{attribute 'qualified_only'}
VAR_GLOBAL CONSTANT
	cuiNrChannel		: UINT	:= 79;
END_VAR

(* stored: Version 1.1.0.1, ProductVersion 3.1.4024.6
   GVL GVL: Id {de6b6213-4d0e-42d5-af64-7295693e9e6d} *)
